FUNCTION_BLOCK FB_ReadCoil
VAR
	fbMBReadCoils : FB_MBReadCoils;
	nReadValue: BYTE;
	
	eReadState : (WAIT, TRIGGER, READ);
	
	fbTrigger : R_TRIG;
END_VAR

fbTrigger();
IF fbTrigger.Q THEN 
	IF eReadState = WAIT THEN
		eReadState := TRIGGER;
	END_IF
END_IF

CASE eReadState OF 
	WAIT:
	//DO
	
	TRIGGER:
	fbMBReadCoils(
 	   sIPAddr  := '10.17.76.191',
       nTCPPort  := 502,
       nUnitID    :=16#FF,
       nQuantity  := 1,
       nMBAddr  := 0,
       cbLength := SIZEOF(nReadValue) ,    
       pDestAddr := ADR(nReadValue),
       bExecute   := TRUE ,
       tTimeout:= ,
       bError =>   ,
       nErrId => ,
       cbRead  =>   );
	
	eReadState := READ;
	
	READ:
	//Wait for the response 
	fbMBReadCoils(bExecute := FALSE);
	IF NOT fbMBReadCoils.bBusy OR fbMBReadCoils.bError THEN
		eReadState:= WAIT;
	END_IF
	
END_CASE

END_FUNCTION_BLOCK

(* stored: Version 1.1.0.1, ProductVersion 3.1.4024.16
   POU FB_ReadCoil: Id {1ccb2c5d-4f5c-44a7-846e-1ec317b1d795}, SpecialFunc None *)
